# EPICS substitutions: modules/event/evrSupport/Db/ioc/IOC-IN20-PM01evr.substitutions
#==============================================================================
#
# Abs:  LCLS EVR IOC records for IN20 PM01
#
# Name: IOC-IN20-PM01evr.substitutions
#
#==============================================================================
#
file evrPMXX.db
{
pattern { DEVICE        }
	{ EVR:IN20:PM01 }
}
